// TIA Portal V17 export
// export: Created 2024-08-09T12:53:22.1452181Z, ExportSetting WithDefaults, DisplayName Totally Integrated Automation Portal, DisplayVersion V17 Update 7, DisplayName TIA Portal Openness, DisplayVersion V17 Update 7, DisplayName TIA Portal Version Control Interface, DisplayVersion V17, DisplayName STEP 7 Professional, DisplayVersion V17 Update 7, DisplayName STEP 7 Safety, DisplayVersion V17 Update 6, DisplayName WinCC Professional, DisplayVersion V17 Update 7
TYPE "S_ChargCompo"
// stored: IsFailsafeCompliant false
   STRUCT
      _Ptzs { ExternalAccessible := 'False'; ExternalVisible := 'False'; ExternalWritable := 'False'} : "S_SuiviCommande";   // adresse zone de suivi de lot
      _Ptcompo { ExternalAccessible := 'False'; ExternalVisible := 'False'; ExternalWritable := 'False'} : "S_Compo_char";   // adresse compo a charger
      _Circuit { ExternalAccessible := 'False'; ExternalVisible := 'False'; ExternalWritable := 'False'} : "S_Circuit";
      _PtChargPont { ExternalAccessible := 'False'; ExternalVisible := 'False'; ExternalWritable := 'False'} : "S_ChargPont";   // Classe chargement pont associ
      _TabCircuitPreremp { ExternalAccessible := 'False'; ExternalVisible := 'False'; ExternalWritable := 'False'} : Array[0.."Nbr_Mob_Circuit"] of "S_Mob_Cir";   // Liste des mobiles a demarrer pour le preremplissage
      _ChargCommun { ExternalAccessible := 'False'; ExternalVisible := 'False'; ExternalWritable := 'False'} : "S_ChargCommun";
      _ListeTaAttAutPreremplissage { ExternalAccessible := 'False'; ExternalVisible := 'False'; ExternalWritable := 'False'} : Array[0.."T_MAX_AMONTAVAL"] of "S_TacheNiv";
      _ListeTaAttAutDemarrage { ExternalAccessible := 'False'; ExternalVisible := 'False'; ExternalWritable := 'False'} : Array[0.."T_MAX_AMONTAVAL"] of "S_TacheNiv";
      _ListeTaAttAttAutVidange { ExternalAccessible := 'False'; ExternalVisible := 'False'; ExternalWritable := 'False'} : Array[0.."T_MAX_AMONTAVAL"] of "S_TacheNiv";
      _ListeTaAttFinLotCharg { ExternalAccessible := 'False'; ExternalVisible := 'False'; ExternalWritable := 'False'} : Array[0.."T_MAX_AMONTAVAL"] of "S_TacheNiv";
      Dial_Def { ExternalAccessible := 'False'; ExternalVisible := 'False'; ExternalWritable := 'False'} : "S_DIALOG_DEF";
      _TpsPicke { ExternalAccessible := 'False'; ExternalVisible := 'False'; ExternalWritable := 'False'} : Date_And_Time;
      _DebutNb { ExternalAccessible := 'False'; ExternalVisible := 'False'; ExternalWritable := 'False'} : Date_And_Time;
      _FiltreNiveauBas { ExternalAccessible := 'False'; ExternalVisible := 'False'; ExternalWritable := 'False'} : Time;   // Filtre niveau bas
      _SavVisCharg { ExternalAccessible := 'False'; ExternalVisible := 'False'; ExternalWritable := 'False'} : Real;   // Sortie analogique commande vis chargement
      _VitFinCharg { ExternalAccessible := 'False'; ExternalVisible := 'False'; ExternalWritable := 'False'} : Real;   // Vitesse vis de chargement en fin de chargement
      _DebitPont { ExternalAccessible := 'False'; ExternalVisible := 'False'; ExternalWritable := 'False'} : Real;   // Debit pont
      _DebitMaxVisCharg { ExternalAccessible := 'False'; ExternalVisible := 'False'; ExternalWritable := 'False'} : Real;   // Debit maximum vis de chargement
      _VitPreremp { ExternalAccessible := 'False'; ExternalVisible := 'False'; ExternalWritable := 'False'} : Real;   // Vitesse vis prremplissage
      _SeuilQteDemCharg { ExternalAccessible := 'False'; ExternalVisible := 'False'; ExternalWritable := 'False'} : Real;   // Seuil quantite sur pont pour demarrer le chargement
      _SeuilQteFinCharg { ExternalAccessible := 'False'; ExternalVisible := 'False'; ExternalWritable := 'False'} : Real;   // Seuil quantite Restante a charger pour augmenter la vitesse des minraux
      _OrigineCharg { ExternalAccessible := 'False'; ExternalVisible := 'False'; ExternalWritable := 'False'} : Int;   // Origine du chargement
      _CptNbTourPreremp { ExternalAccessible := 'False'; ExternalVisible := 'False'; ExternalWritable := 'False'} : Int;   // Compteur nombre de tour pour preremplissage
      _MbTamis { ExternalAccessible := 'False'; ExternalVisible := 'False'; ExternalWritable := 'False'} : Int;
      _MobDeasserv { ExternalAccessible := 'False'; ExternalVisible := 'False'; ExternalWritable := 'False'} : Int;
      _NbTourPreremp { ExternalAccessible := 'False'; ExternalVisible := 'False'; ExternalWritable := 'False'} : Int;   // Nombre de tour pour preremplissage
      _VitMinVisCharg { ExternalAccessible := 'False'; ExternalVisible := 'False'; ExternalWritable := 'False'} : Int;   // Vitesse minimum vis de chargement
      _VitMaxVisCharg { ExternalAccessible := 'False'; ExternalVisible := 'False'; ExternalWritable := 'False'} : Int;   // Vitesse maximum vis de chargement
      _SRazNbTourPreremp { ExternalAccessible := 'False'; ExternalVisible := 'False'; ExternalWritable := 'False'} : USInt;   // Sortie remise a 0 compteur nombre de tour pour preremplissage
      _NumPont { ExternalAccessible := 'False'; ExternalVisible := 'False'; ExternalWritable := 'False'} : USInt;   // Num Pont
      _LectChute { ExternalAccessible := 'False'; ExternalVisible := 'False'; ExternalWritable := 'False'} : SInt;   // Lecture colonne de chute en base
      _DebitPontMini { ExternalAccessible := 'False'; ExternalVisible := 'False'; ExternalWritable := 'False'} : SInt;   // Dbit minimum du pont pour gestion vitesse incorpo avec dbit du pont
      _NoCompo { ExternalAccessible := 'False'; ExternalVisible := 'False'; ExternalWritable := 'False'} : SInt;   // No de compansant
      _ArrImmMemeProd { ExternalAccessible := 'False'; ExternalVisible := 'False'; ExternalWritable := 'False'} : Bool;   // Possibilite Arret immediat circuit
      _SuspCircuit { ExternalAccessible := 'False'; ExternalVisible := 'False'; ExternalWritable := 'False'} : Bool;   // Suspension circuit
      _ValidPoidsTheo { ExternalAccessible := 'False'; ExternalVisible := 'False'; ExternalWritable := 'False'} : Bool;   // Flag validation mouvement poids thorique
      _GestVitDebitTheo { ExternalAccessible := 'False'; ExternalVisible := 'False'; ExternalWritable := 'False'} : Bool;   // Gestion vitesse de chargement sur dbit pont thorique
      _PrerempEc { ExternalAccessible := 'False'; ExternalVisible := 'False'; ExternalWritable := 'False'} : Bool;
      _NivBasTremie { ExternalAccessible := 'False'; ExternalVisible := 'False'; ExternalWritable := 'False'} : Bool;   // Niveau bas tremie
      _PresenceCapNivBasTremie { ExternalAccessible := 'False'; ExternalVisible := 'False'; ExternalWritable := 'False'} : Bool;   // Presence cap Niveau bas tremie
      _EPmMobCharg { ExternalAccessible := 'False'; ExternalVisible := 'False'; ExternalWritable := 'False'} : Bool;   // Passage matiere pour preremplissage
      _EPmPreremp { ExternalAccessible := 'False'; ExternalVisible := 'False'; ExternalWritable := 'False'} : Bool;   // Passage matiere pour preremplissage
      _Vibreur { ExternalAccessible := 'False'; ExternalVisible := 'False'; ExternalWritable := 'False'} : Bool;   // Sortie vibreur
   END_STRUCT;
END_TYPE
